KUKA KRL data list: global_eki.dat

&ACCESS RVO
&REL 49
defdat global_eki public
   global bool ROBOT_STOPPED
   global INT META_VELOCITY_OVERRIDE
enddat
